FUNCTION_BLOCK FB_ContextBuilder IMPLEMENTS I_ContextBuilder
VAR_INPUT
END_VAR
VAR_OUTPUT
END_VAR
VAR
END_VAR

{warning 'add method implementation '}
METHOD WithContextInt : I_ContextBuilder
VAR_INPUT
	sName	: Tc2_System.T_MaxString;
	nValue	: INT;
END_VAR
END_METHOD

END_FUNCTION_BLOCK

(* stored: Version 1.1.0.1, ProductVersion 3.1.4024.0
   POU FB_ContextBuilder: Id {7f1d5e34-ea3b-4ad5-887e-933d0a5923d7}, SpecialFunc None
   Method WithContextInt: Id {fb2119ae-4050-4e81-8815-a8079d098669} *)
